// TIA Portal V18 program export: 2 tag tables, 0 data types, 2 data blocks, 1 code blocks (in call order from the OBs), 0 instance data blocks

VAR_GLOBAL   // PLC tag table "AI_Tags"
   MB_Server_NDR AT %M10.0 : Bool;   // MB_Server_NDR Modbus Tag
   MB_Server_DR AT %M10.1 : Bool;   // MB_Server_DR Modbus Tag
   MB_Server_Error AT %M10.2 : Bool;   // MB_Server_Error Modbus Tag
   MB_Server_Status AT %MW12 : Word;   // MB_Server_Status Modbus Tag
END_VAR

VAR_GLOBAL   // PLC tag table "Default tag table"
   System_Byte AT %MB1 : Byte;
   FirstScan AT %M1.0 : Bool;
   DiagStatusUpdate AT %M1.1 : Bool;
   AlwaysTRUE AT %M1.2 : Bool;
   AlwaysFALSE AT %M1.3 : Bool;
   Clock_Byte AT %MB0 : Byte;
   Clock_10Hz AT %M0.0 : Bool;
   Clock_5Hz AT %M0.1 : Bool;
   "Clock_2.5Hz" AT %M0.2 : Bool;
   Clock_2Hz AT %M0.3 : Bool;
   "Clock_1.25Hz" AT %M0.4 : Bool;
   Clock_1Hz AT %M0.5 : Bool;
   "Clock_0.625Hz" AT %M0.6 : Bool;
   "Clock_0.5Hz" AT %M0.7 : Bool;
END_VAR

DATA_BLOCK "DB_MB_Server_Conn"   // DB13
TITLE = DB_MB_Server_Conn
{ S7_Optimized_Access := 'FALSE' }
VERSION : 0.1
// DB communication via Modbus TCP
// stored: AutoNumber false, DBAccessibleFromOPCUA true, IsOnlyStoredInLoadMemory false, IsWriteProtectedInAS false
   VAR
      MB_TCP_SERVER : TCON_IP_v4;
   END_VAR
BEGIN
END_DATA_BLOCK

DATA_BLOCK "DB_Modbus_Holding_Register"   // DB12
TITLE = DB_Modbus_Holding_Register
{ S7_Optimized_Access := 'FALSE' }
VERSION : 0.1
// DB communication via Modbus TCP
// stored: AutoNumber false, DBAccessibleFromOPCUA true, IsOnlyStoredInLoadMemory false, IsWriteProtectedInAS false
   VAR
      CmdSeq : Int;
      CmdBools : Int;
      Heartbeat_Client : Int;
      AckSeq : Int;
      StatusBools : Int;
      State : Int;
      PID_Bon4_SP : Real;
      PID_Bon4_PV : Real;
      PID_Bon4_CV : Real;
      Heartbeat_Server : Int;
   END_VAR
BEGIN
END_DATA_BLOCK

ORGANIZATION_BLOCK "Main"   // OB1, LAD, ProgramCycle
TITLE = "Main Program Sweep (Cycle)"
{ S7_Optimized_Access := 'TRUE' }
VERSION : 0.1
// stored: AutoNumber true, IsIECCheckEnabled false, SetENOAutomatically false
   VAR_INPUT
      Initial_Call : Bool;   // Initial call of this OB
      Remanence : Bool;   // =True, if remanent data are available
   END_VAR
BEGIN

REGION Network 1
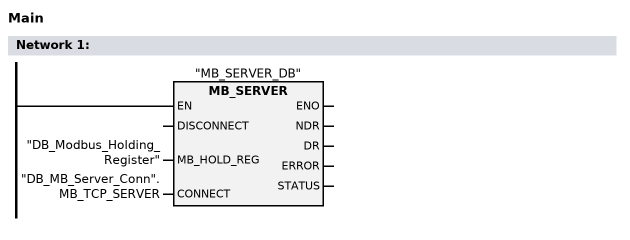
   RUNG wire#powerrail
      "MB_SERVER_DB".MB_SERVER(DISCONNECT :=, MB_HOLD_REG := "DB_Modbus_Holding_Register", CONNECT := "DB_MB_Server_Conn".MB_TCP_SERVER, NDR =>, DR =>, ERROR =>, STATUS =>)
   END_RUNG
   // the same network as SCL:
   "MB_SERVER_DB"(MB_HOLD_REG := "DB_Modbus_Holding_Register", CONNECT := "DB_MB_Server_Conn".MB_TCP_SERVER);   // MB_SERVER
END_REGION
END_ORGANIZATION_BLOCK
